// TIA Portal V19 export
FUNCTION_BLOCK "AFB_Totalizer"   // FB3, LAD
{ S7_Optimized_Access := 'TRUE' }
// stored: MemoryReserve 100, SetENOAutomatically false
   VAR_INPUT
      inputVolume { ExternalAccessible := 'False'; ExternalVisible := 'False'; ExternalWritable := 'False'} : Real;
      startBtn { ExternalAccessible := 'False'; ExternalVisible := 'False'; ExternalWritable := 'False'} : Bool;
      stopBtn { ExternalAccessible := 'False'; ExternalVisible := 'False'; ExternalWritable := 'False'} : Bool;
   END_VAR
   VAR_OUTPUT
      addedVolume { ExternalAccessible := 'False'; ExternalVisible := 'False'; ExternalWritable := 'False'} : Real;
      tempCount { ExternalAccessible := 'False'; ExternalVisible := 'False'; ExternalWritable := 'False'} : Bool;
   END_VAR
   VAR
      previousVolume { ExternalAccessible := 'False'; ExternalVisible := 'False'; ExternalWritable := 'False'} : Real;
      Start_Trigger { S7_SetPoint := 'True'} : R_TRIG;
      Strop_Trigger { S7_SetPoint := 'True'} : R_TRIG;
   END_VAR
BEGIN

REGION Network 1
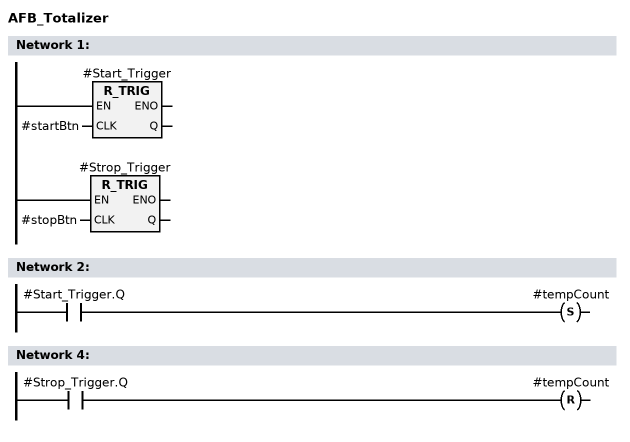
   RUNG wire#powerrail
      #Start_Trigger.R_TRIG(CLK := #startBtn, Q =>)
   END_RUNG
   RUNG wire#powerrail
      #Strop_Trigger.R_TRIG(CLK := #stopBtn, Q =>)
   END_RUNG
   // the same network as SCL:
   #Start_Trigger(CLK := #startBtn);   // R_TRIG
   #Strop_Trigger(CLK := #stopBtn);   // R_TRIG
END_REGION

REGION Network 2
   RUNG wire#powerrail
      Contact( #Start_Trigger.Q )
      S_Coil( #tempCount )
   END_RUNG
   // the same network as SCL:
   IF #Start_Trigger.Q THEN #tempCount := TRUE; END_IF;
END_REGION

REGION Network 3 (SCL)

   IF #startBtn THEN
       #previousVolume := #inputVolume;
   END_IF;


   IF #tempCount THEN

       #addedVolume := #inputVolume - #previousVolume;
       ;
   ELSE
       #addedVolume := 0 ;
   END_IF;
END_REGION

REGION Network 4
   RUNG wire#powerrail
      Contact( #Strop_Trigger.Q )
      R_Coil( #tempCount )
   END_RUNG
   // the same network as SCL:
   IF #Strop_Trigger.Q THEN #tempCount := FALSE; END_IF;
END_REGION
END_FUNCTION_BLOCK
